Omron CX-Programmer project NewProject (CX-Programmer 9.50)

# PLC NewPLC1: CJ1M CPU21

## Global symbols (name address type ; comment)
0.00 BOOL  ; PB ON
0.01 BOOL  ; PB OFF
1.00 BOOL  ; LED ON
1.01 BOOL  ; LED OFF
2001 CHANNEL  ; output analog 1
2005 CHANNEL  ; input analog 1
2006 CHANNEL  ; input analog 2
D0 CHANNEL  ; nilai sensor/nilai tujuan terkecil [RTD]
D1 CHANNEL  ; nilai asal terkecil [RTD]
D10 CHANNEL  ; hasil SCL (BCD) [ultrasonic]
D11 CHANNEL  ; hasil SCL (BIN) [ultrasonic]
D12 CHANNEL  ; konversi output (REAL ke BIN)
D13 CHANNEL  ; nilai terkecil tujuan [motor fan]
D14 CHANNEL  ; nilai asal terkecil [motor fan]
D15 CHANNEL  ; nilai tujuan terbesar [motor fan]
D16 CHANNEL  ; nilai asal terbesar [motor fan]
D17 CHANNEL  ; Hasil SCL (BCD) [motorfan]
D18 CHANNEL  ; hasil SCL (BIN) [motorfan]
D19 CHANNEL  ; nilai terkecil tujuan volt [RTD]
D2 CHANNEL  ; nilai tujuan terbesar [RTD]
D20 CHANNEL  ; nilai terkecil resolusi volt [RTD]
D21 CHANNEL  ; nilai terbesar tujuan volt [RTD]
D22 CHANNEL  ; nilai terbesar resolusi volt [RTD]
D23 CHANNEL  ; hasil SCL volt (BCD) [RTD]
D24 CHANNEL  ; hasil SCL volt (BIN) [RTD]
D25 CHANNEL  ; nilai SCL (REAL) [RTD]
D27 CHANNEL  ; hasil SCL (REAL) [ultrasonic]
D29 CHANNEL  ; Output Motor fan (REAL)
D3 CHANNEL  ; nilai asal terbesar [RTD]
D32 CHANNEL  ; nilai terkecil tujuan arus [ultrasonic]
D33 CHANNEL  ; nilai terkecil resolusi arus [ultrasonic]
D34 CHANNEL  ; nilai terbesar tujuan arus [ultrasonic]
D35 CHANNEL  ; nilai terbesar resolusi arus [ultrasonic]
D36 CHANNEL  ; hasil SCL arus (BCD) [ultrasonic]
D37 CHANNEL  ; nilai SCL arus (BIN) [ultrasonic]
D38 CHANNEL  ; nilai terkecil tujuan volt [motor fan]
D39 CHANNEL  ; nilai terkecil resolusi volt [motor fan]
D4 CHANNEL  ; nilai SCL (BCD) [RTD]
D40 CHANNEL  ; nilai terbesar tujuan volt [motor fan]
D41 CHANNEL  ; nilai terbesar resolusi volt [motor fan]
D42 CHANNEL  ; hasil SCL volt (BCD) [motor fan]
D43 CHANNEL  ; hasil SCL volt (BIN) [motor fan]
D5 CHANNEL  ; nilai SCL (BIN) [RTD]
D6 CHANNEL  ; nilai sensor/nilai tujuan terkecil [ultrasonic]
D7 CHANNEL  ; nilai asal terkecil [ultrasonic]
D8 CHANNEL  ; nilai tujuan terbesar [ultrasonic]
D9 CHANNEL  ; nilai asal terbesar [ultrasonic]
Fuzzy fuzychiller
fuzy fuzychiller

## Program NewProgram1 (cyclic task 0)

### Section Section1

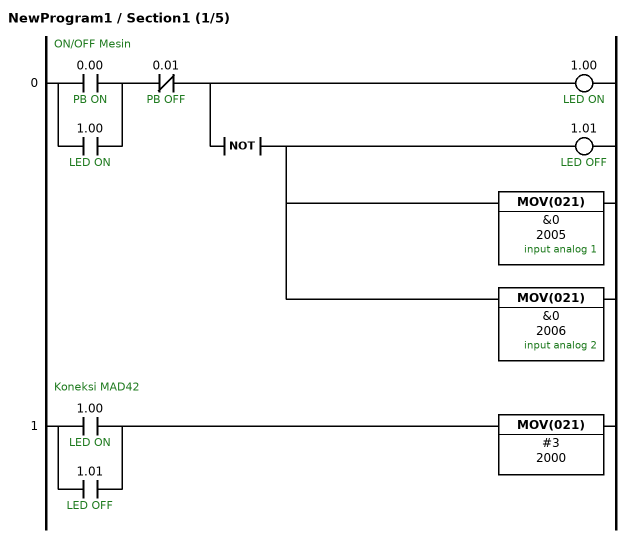
; rung 0: ON/OFF Mesin
LD 0.00  ; PB ON
OR 1.00  ; LED ON
ANDNOT 0.01  ; PB OFF
OUT 1.00  ; LED ON
NOT(520)
OUT 1.01  ; LED OFF
MOV(021) &0 2005  ; input analog 1
MOV(021) &0 2006  ; input analog 2
; rung 1: Koneksi MAD42
LD 1.00  ; LED ON
OR 1.01  ; LED OFF
MOV(021) #3 2000

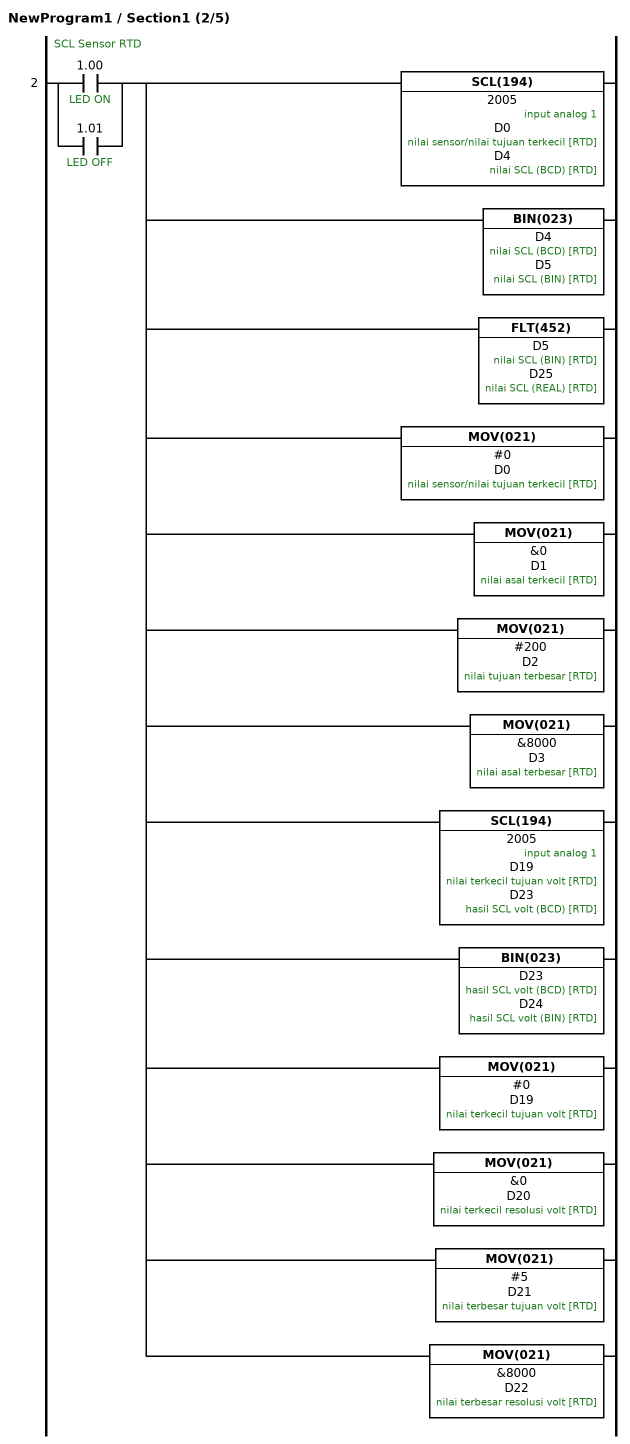
; rung 2: SCL Sensor RTD
LD 1.00  ; LED ON
OR 1.01  ; LED OFF
SCL(194) 2005 D0 D4  ; input analog 1, nilai sensor/nilai tujuan terkecil [RTD], nilai SCL (BCD) [RTD]
BIN(023) D4 D5  ; nilai SCL (BCD) [RTD], nilai SCL (BIN) [RTD]
FLT(452) D5 D25  ; nilai SCL (BIN) [RTD], nilai SCL (REAL) [RTD]
MOV(021) #0 D0  ; nilai sensor/nilai tujuan terkecil [RTD]
MOV(021) &0 D1  ; nilai asal terkecil [RTD]
MOV(021) #200 D2  ; nilai tujuan terbesar [RTD]
MOV(021) &8000 D3  ; nilai asal terbesar [RTD]
SCL(194) 2005 D19 D23  ; input analog 1, nilai terkecil tujuan volt [RTD], hasil SCL volt (BCD) [RTD]
BIN(023) D23 D24  ; hasil SCL volt (BCD) [RTD], hasil SCL volt (BIN) [RTD]
MOV(021) #0 D19  ; nilai terkecil tujuan volt [RTD]
MOV(021) &0 D20  ; nilai terkecil resolusi volt [RTD]
MOV(021) #5 D21  ; nilai terbesar tujuan volt [RTD]
MOV(021) &8000 D22  ; nilai terbesar resolusi volt [RTD]

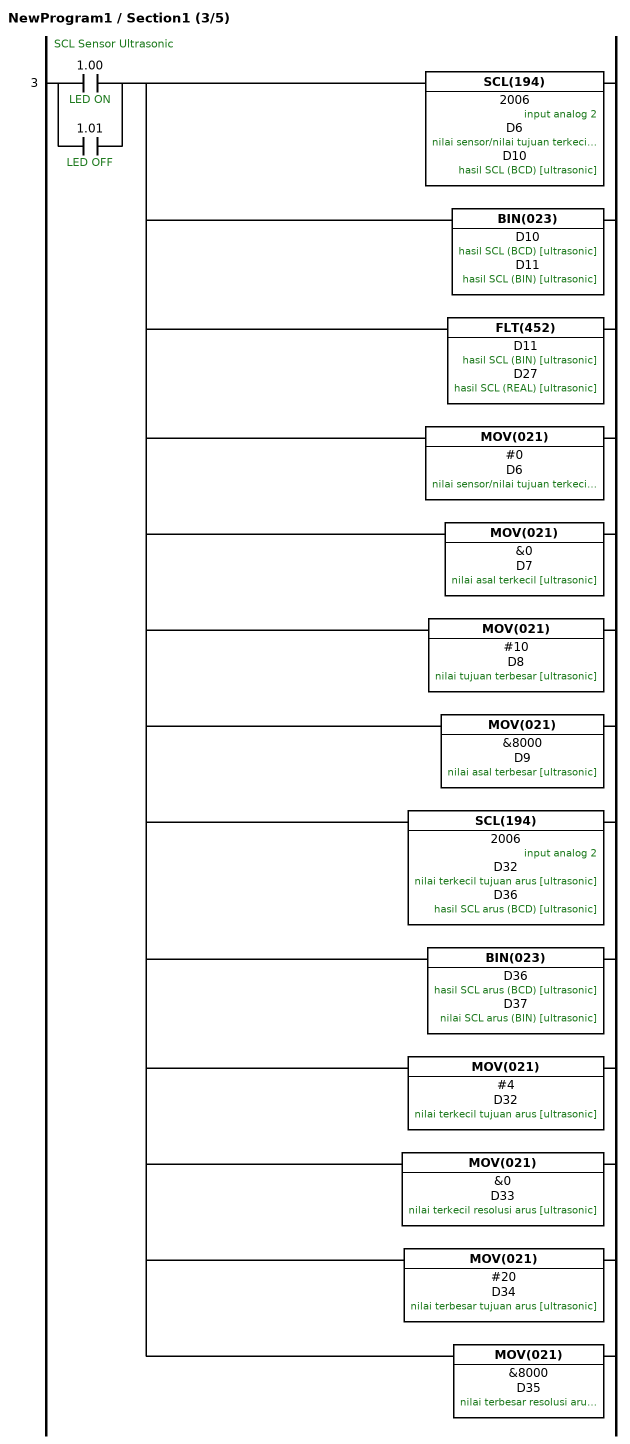
; rung 3: SCL Sensor Ultrasonic
LD 1.00  ; LED ON
OR 1.01  ; LED OFF
SCL(194) 2006 D6 D10  ; input analog 2, nilai sensor/nilai tujuan terkecil [ultrasonic], hasil SCL (BCD) [ultrasonic]
BIN(023) D10 D11  ; hasil SCL (BCD) [ultrasonic], hasil SCL (BIN) [ultrasonic]
FLT(452) D11 D27  ; hasil SCL (BIN) [ultrasonic], hasil SCL (REAL) [ultrasonic]
MOV(021) #0 D6  ; nilai sensor/nilai tujuan terkecil [ultrasonic]
MOV(021) &0 D7  ; nilai asal terkecil [ultrasonic]
MOV(021) #10 D8  ; nilai tujuan terbesar [ultrasonic]
MOV(021) &8000 D9  ; nilai asal terbesar [ultrasonic]
SCL(194) 2006 D32 D36  ; input analog 2, nilai terkecil tujuan arus [ultrasonic], hasil SCL arus (BCD) [ultrasonic]
BIN(023) D36 D37  ; hasil SCL arus (BCD) [ultrasonic], nilai SCL arus (BIN) [ultrasonic]
MOV(021) #4 D32  ; nilai terkecil tujuan arus [ultrasonic]
MOV(021) &0 D33  ; nilai terkecil resolusi arus [ultrasonic]
MOV(021) #20 D34  ; nilai terbesar tujuan arus [ultrasonic]
MOV(021) &8000 D35  ; nilai terbesar resolusi arus [ultrasonic]

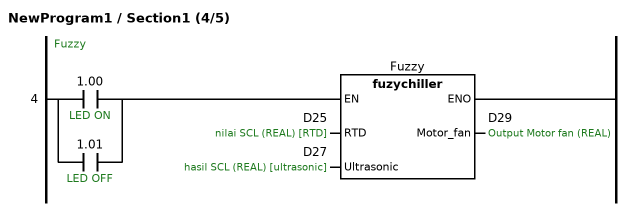
; rung 4: Fuzzy
LD 1.00  ; LED ON
OR 1.01  ; LED OFF
CALL Fuzzy : fuzychiller (RTD := D25, Ultrasonic := D27, Motor_fan => D29)  ; nilai SCL (REAL) [RTD], hasil SCL (REAL) [ultrasonic], Output Motor fan (REAL)

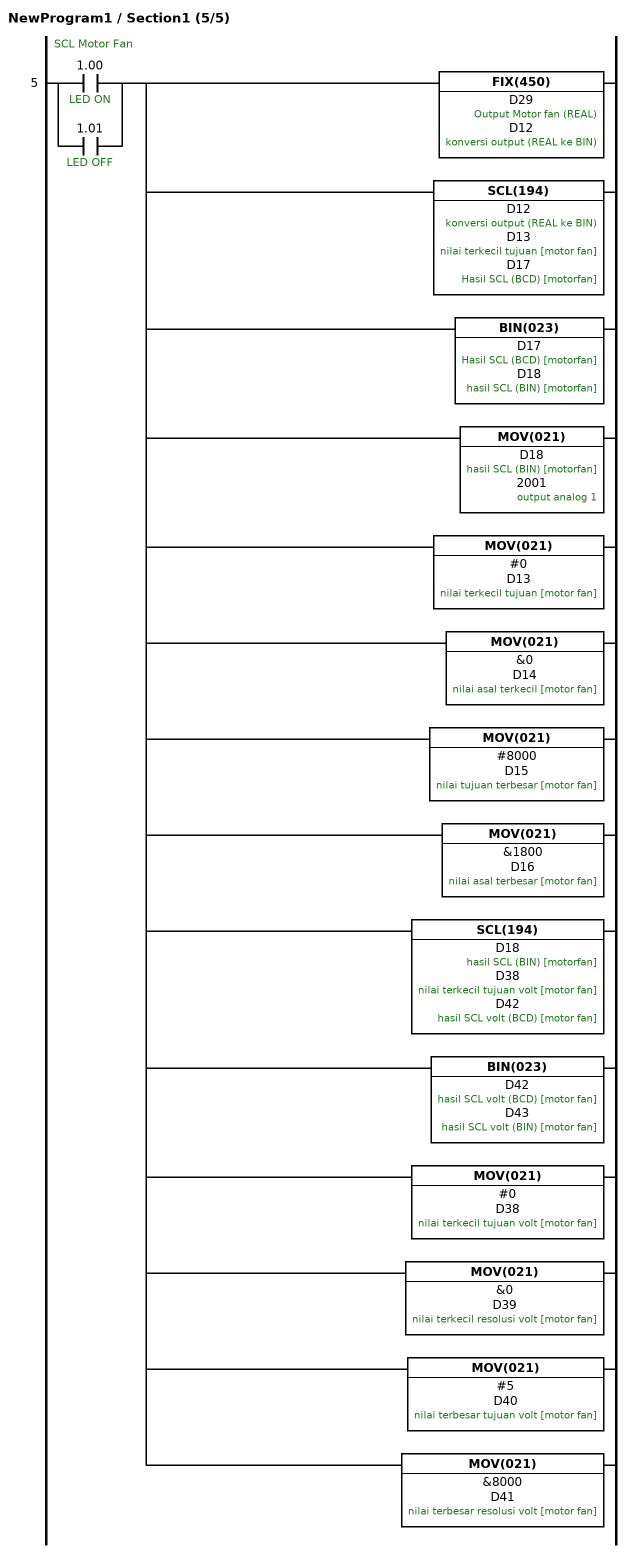
; rung 5: SCL Motor Fan
LD 1.00  ; LED ON
OR 1.01  ; LED OFF
FIX(450) D29 D12  ; Output Motor fan (REAL), konversi output (REAL ke BIN)
SCL(194) D12 D13 D17  ; konversi output (REAL ke BIN), nilai terkecil tujuan [motor fan], Hasil SCL (BCD) [motorfan]
BIN(023) D17 D18  ; Hasil SCL (BCD) [motorfan], hasil SCL (BIN) [motorfan]
MOV(021) D18 2001  ; hasil SCL (BIN) [motorfan], output analog 1
MOV(021) #0 D13  ; nilai terkecil tujuan [motor fan]
MOV(021) &0 D14  ; nilai asal terkecil [motor fan]
MOV(021) #8000 D15  ; nilai tujuan terbesar [motor fan]
MOV(021) &1800 D16  ; nilai asal terbesar [motor fan]
SCL(194) D18 D38 D42  ; hasil SCL (BIN) [motorfan], nilai terkecil tujuan volt [motor fan], hasil SCL volt (BCD) [motor fan]
BIN(023) D42 D43  ; hasil SCL volt (BCD) [motor fan], hasil SCL volt (BIN) [motor fan]
MOV(021) #0 D38  ; nilai terkecil tujuan volt [motor fan]
MOV(021) &0 D39  ; nilai terkecil resolusi volt [motor fan]
MOV(021) #5 D40  ; nilai terbesar tujuan volt [motor fan]
MOV(021) &8000 D41  ; nilai terbesar resolusi volt [motor fan]

### Section END
; rung 0
END(001)

## Function block fuzychiller
VAR_INPUT
  RTD : REAL;
  Ultrasonic : REAL;
END_VAR
VAR_OUTPUT
  Motor_fan : REAL;
END_VAR
VAR
  Slow : REAL := 500.0;
  High : REAL := 1800.0;
  Med : REAL := 1000.0;
  rule9 : REAL;
  rule8 : REAL;
  rule7 : REAL;
  rule6 : REAL;
  rule5 : REAL;
  rule4 : REAL;
  rule3 : REAL;
  rule2 : REAL;
  rule1 : REAL;
  US_hi : REAL;
  US_med : REAL;
  US_low : REAL;
  RTD_hot : REAL;
  RTD_med : REAL;
  RTD_cold : REAL;
END_VAR
(*RTD PT100 Fuzzyfication*)

IF RTD <= 20,0 THEN
	RTD_cold := 1,0;
	RTD_med :=  0,0;
	RTD_hot :=  0,0;
	
ELSIF RTD > 20,0 AND RTD < 30,0 THEN
	RTD_cold :=  (30,0-RTD)/(30,0-20,0);
	RTD_med :=  (RTD-20,0)/(30,0-20,0);
	RTD_hot :=  0,0;
	
ELSIF RTD = 30,0 THEN
	RTD_cold :=  0,0;
	RTD_med :=  1,0;
	RTD_hot :=  0,0;
	
ELSIF RTD > 30,0 AND RTD < 40,0 THEN
	RTD_cold :=  0,0;
	RTD_med :=  (40,0 - RTD)/(40,0-30,0);
	RTD_hot :=  (RTD-30,0)/(40,0-30,0);
	
ELSIF RTD >= 40,0 THEN
	RTD_cold :=  0,0;
	RTD_med :=  0,0;
	RTD_hot :=  1,0;
END_IF;

(*Ultrasonic Fuzzyfication*)

IF Ultrasonic <= 3,0 THEN
	US_low :=  1,0;
	US_med :=  0,0;
	US_hi :=  0,0;
	
ELSIF Ultrasonic > 3,0 AND Ultrasonic < 5,0 THEN
	US_low :=  (5,0 - Ultrasonic)/(5,0-3,0);
	US_med :=  (Ultrasonic - 3,0)/(5,0-3,0);
	US_hi :=  0,0;
	
ELSIF Ultrasonic = 5,0 THEN
	US_low :=  0,0;
	US_med :=  1,0;
	US_hi :=  0,0;

ELSIF Ultrasonic > 5,0 AND Ultrasonic < 7,0 THEN
	US_low :=  0,0;
	US_med :=  (7,0 - Ultrasonic)/(7,0-5,0);
	US_hi :=  (Ultrasonic-5,0)/(7,0-5,0);
	
ELSIF Ultrasonic >= 7,0 THEN
	US_low :=  0,0;
	US_med :=  0,0;
	US_hi :=  1,0;
END_IF;

(*Rules*)
rule1 :=  MIN(RTD_cold,US_low);
rule2 :=  MIN(RTD_cold,US_med);
rule3 :=  MIN(RTD_cold, US_hi);
rule4 :=  MIN(RTD_med, US_low);
rule5 :=  MIN(RTD_med, US_med);
rule6 :=  MIN(RTD_med, US_hi);
rule7 :=  MIN(RTD_hot, US_low);
rule8 :=  MIN(RTD_hot, US_med);
rule9 :=  MIN(RTD_hot, US_hi);

(*Defuzification of Weight Average*)
Motor_fan :=  ((rule1*Slow) + (rule2*Slow) + (rule3* Med) + (rule4*Slow) + (rule5*Med) + (rule6*Med) + (rule7*Med) + (rule8*High) + (rule9*High)) / (rule1+rule2+rule3+rule4+rule5+rule6+rule7+rule8+rule9);